Fanuc KAREL source: kt00700.KL

-- PROVISIONAL review KL for V1013-1; original PC SHA256 bdbe7af0bcc5485c2a3010b1249e1b1f2a3ef81cadfc17869ae7acd00fab047a
-- Incomplete behavior may be omitted. Consult companion uncertainty JSON. Do not deploy.
PROGRAM KT00700
%NOLOCKGROUP
VAR
  OUT : INTEGER
-- UNRESOLVED_DECL C1 type=00001c
-- UNRESOLVED_DECL C2 type=00001c
BEGIN
  -- UNRESOLVED_PC offsets 5-15; opcodes 9D,22,A5
  -- UNRESOLVED_PC offsets 20-30; opcodes 9C,22,A5
  -- UNRESOLVED_PC offsets 35-45; opcodes 9D,22,A5
  -- UNRESOLVED_PC offsets 50-60; opcodes 9C,22,A5
  -- UNRESOLVED_PC offsets 65-77; opcodes 21,23
  -- UNRESOLVED_PC offsets 82-86; opcodes 7F
END KT00700
